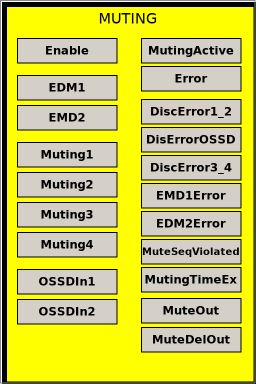
VISUALIZATION V_PH_MUTING  // 256x384
VAR_INPUT
	stSafetyMuting				:ST_SAFETY_FBMUTING;
END_VAR
    Rectangle (2,2 256x384), colour toggle: stSafetyMuting.bGeneralError
    RoundedRectangle (17,142 100x25), "Muting1", colour toggle: stSafetyMuting.uStatus.stStatusWords.wInputs.8
    RoundedRectangle (17,38 100x25), "Enable", colour toggle: stSafetyMuting.uStatus.stStatusWords.wInputs.0
    RoundedRectangle (17,105 100x25), "EMD2", colour toggle: stSafetyMuting.uStatus.stStatusWords.wInputs.2
    RoundedRectangle (17,172 100x25), "Muting2", colour toggle: stSafetyMuting.uStatus.stStatusWords.wInputs.9
    RoundedRectangle (17,202 100x25), "Muting3", colour toggle: stSafetyMuting.uStatus.stStatusWords.wInputs.10
    RoundedRectangle (17,299 100x25), "OSSDIn2", colour toggle: stSafetyMuting.uStatus.stStatusWords.wInputs.13
    RoundedRectangle (17,232 100x25), "Muting4", colour toggle: stSafetyMuting.uStatus.stStatusWords.wInputs.11
    RoundedRectangle (17,269 100x25), "OSSDIn1", colour toggle: stSafetyMuting.uStatus.stStatusWords.wInputs.12
    RoundedRectangle (17,75 100x25), "EDM1", colour toggle: stSafetyMuting.uStatus.stStatusWords.wInputs.1
    Label (5,6 246x25), "MUTING"
    RoundedRectangle (141,38 100x25), "MutingActive", colour toggle: stSafetyMuting.uStatus.stStatusWords.wOutputs.1
    RoundedRectangle (141,66 100x25), "Error", colour toggle: stSafetyMuting.uStatus.stStatusWords.wOutputs.0
    RoundedRectangle (141,298 100x25), "MuteOut", colour toggle: stSafetyMuting.uStatus.stStatusWords.wOutputs.2
    RoundedRectangle (141,327 100x25), "MuteDelOut", colour toggle: stSafetyMuting.uStatus.stStatusWords.wOutputs.3
    RoundedRectangle (141,127 100x25), "DisErrorOSSD", colour toggle: stSafetyMuting.uStatus.stStatusWords.wDiagnosis.1, invisible if: NOT stSafetyMuting.uStatus.stStatusWords.wDiagnosis.1
    RoundedRectangle (141,183 100x25), "EMD1Error", colour toggle: stSafetyMuting.uStatus.stStatusWords.wDiagnosis.4, invisible if: NOT stSafetyMuting.uStatus.stStatusWords.wDiagnosis.4
    RoundedRectangle (141,99 100x25), "DiscError1_2", colour toggle: stSafetyMuting.uStatus.stStatusWords.wDiagnosis.0, invisible if: NOT stSafetyMuting.uStatus.stStatusWords.wDiagnosis.0
    RoundedRectangle (141,155 100x25), "DiscError3_4", colour toggle: stSafetyMuting.uStatus.stStatusWords.wDiagnosis.2, invisible if: NOT stSafetyMuting.uStatus.stStatusWords.wDiagnosis.2
    RoundedRectangle (141,267 100x25), "MutingTimeEx", colour toggle: stSafetyMuting.uStatus.stStatusWords.wDiagnosis.7, invisible if: NOT stSafetyMuting.uStatus.stStatusWords.wDiagnosis.7
    RoundedRectangle (141,211 100x25), "EDM2Error", colour toggle: stSafetyMuting.uStatus.stStatusWords.wDiagnosis.5, invisible if: NOT stSafetyMuting.uStatus.stStatusWords.wDiagnosis.5
    RoundedRectangle (141,239 100x25), "MuteSeqViolated", colour toggle: stSafetyMuting.uStatus.stStatusWords.wDiagnosis.6, invisible if: NOT stSafetyMuting.uStatus.stStatusWords.wDiagnosis.6
    Textfield (17,354 234x25), text list: 'TL_FbStateMUTING', text index: stSafetyMuting.eState
END_VISUALIZATION

(* stored: Version 1.1.0.1, ProductVersion 3.1.4024.4
   Visu V_PH_MUTING: Id {4b86b0b6-bc48-4e8a-97da-41fa816a98f3} *)
